Fanuc KAREL source: kb00183.KL

-- PROVISIONAL review KL for V1013-1; original PC SHA256 0ab3d37ea68d1540c0ca6151cf42f434f81c5cfc427ca3598232d085faa00029
-- Incomplete behavior may be omitted. Consult companion uncertainty JSON. Do not deploy.
PROGRAM KB00183
%NOLOCKGROUP
BEGIN
  -- UNRESOLVED_PC offsets 5-12; opcodes 9D,23
  -- UNRESOLVED_PC offsets 17-24; opcodes 9D,23
  -- UNRESOLVED_PC offsets 29-36; opcodes 9D,23
  -- UNRESOLVED_PC offsets 41-77; opcodes 27,22,22,22,1C,22,27,9D,31
  -- UNRESOLVED_PC offsets 82-86; opcodes 7F
END KB00183
